PROGRAM MAIN

SendMessage();
ConfirmableAlarmWithArguments();
AlarmWithCustomSourceInfo();

END_PROGRAM

(* stored: Version 1.1.0.1, ProductVersion 3.1.4024.3
   POU MAIN: Id {9ae84a09-de24-4b52-a2ed-2baa5985f4b1}, SpecialFunc None *)
